FUNCTION_BLOCK ASTORAGE_MUX (* Composite FB wrapping other FBs *)
  (* Standard: 61499-2 *)
  (* Version 0.0, 2008-07-10, 4DIAC-IDE, 4DIAC-Consortium *)
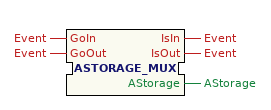
  EVENT_INPUT
    GoIn; (* Confirmation from Plug *)
    GoOut;
  END_EVENT
  EVENT_OUTPUT
    IsIn; (* Request from Socket *)
    IsOut; (* Response from Socket *)
  END_EVENT
  PLUGS
    AStorage : AStorage;
  END_PLUGS
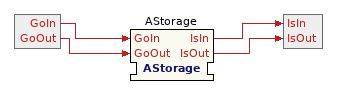
  EVENT_CONNECTIONS
    GoIn TO AStorage.GoIn;
    GoOut TO AStorage.GoOut;
    AStorage.IsIn TO IsIn;
    AStorage.IsOut TO IsOut;
  END_CONNECTIONS
END_FUNCTION_BLOCK
